(* IEC 61131-3 sources: pandora/pandora/aws-platform-main/aws-platform-main/src/Io, 9 files *)

(* ---- Io.st ---- *)
USING Esab.Io;

NAMESPACE Esab.Io

    CLASS ABSTRACT Input
        VAR PUBLIC
            Id : UINT;
            /// The endianness of the read value.
            /// If this is "little" it will be converted to big for use in the PLC-program
            Endianness : Endianness := Endianness#Big;
        END_VAR

        VAR PROTECTED
            _inputChangedHandler : InputChangedListener;
        END_VAR

        METHOD PUBLIC SetChangedHandler
            VAR_INPUT
                handler : InputChangedListener;
            END_VAR

            _inputChangedHandler := handler;
        END_METHOD

        METHOD PUBLIC ABSTRACT HasChanged : BOOL
        END_METHOD
    END_CLASS

    CLASS Output
        VAR PUBLIC
            /// The endianness that the target value is expected to have by the consumer of the output.
            Endianness : Endianness := Endianness#Big;
        END_VAR
    END_CLASS

    INTERFACE InputChangedListener
        METHOD InputChanged
            VAR_INPUT
                input : REF_TO Input;
            END_VAR
        END_METHOD
    END_INTERFACE

    TYPE
        /// Used in Inputs and Outputs to convert endianness properly.
        /// The PLC uses big endian, while data coming from some outside source may be little.
        Endianness : INT(Big := 0, Little := 1);
    END_TYPE

END_NAMESPACE

(* ---- Digital.st ---- *)
NAMESPACE Esab.Io

    INTERFACE IDigitalInput
        /// Reads a new value
        METHOD Read
            VAR_INPUT
                value : BOOL;
            END_VAR
        END_METHOD

        /// Returns the last value read
        METHOD GetValue : BOOL
        END_METHOD

        /// Returns TRUE if the input experienced a rising edge
        METHOD RisingEdge : BOOL
        END_METHOD

        /// Returns TRUE if the input experienced a falling edge
        METHOD FallingEdge : BOOL
        END_METHOD
    END_INTERFACE

    INTERFACE IDigitalOutput
        /// Writes the value to the output
        METHOD Write
            VAR_OUTPUT
                value : BOOL;
            END_VAR
        END_METHOD

        /// Sets the current value to the given value
        METHOD SetValue
            VAR_INPUT
                value: BOOL;
            END_VAR
        END_METHOD

        /// Sets the current value to TRUE
        METHOD Set
        END_METHOD

        /// Reset the current value to FALSE
        METHOD Reset
        END_METHOD

        /// Toggles the current value
        METHOD Toggle
        END_METHOD
    END_INTERFACE

    CLASS DigitalInput EXTENDS Input IMPLEMENTS IDigitalInput
        VAR PRIVATE
            _currentValue : BOOL;
            _lastValue : BOOL;
        END_VAR

        METHOD PUBLIC Read
            VAR_INPUT
                value : BOOL;
            END_VAR

            _lastValue := _currentValue;
            _currentValue := value;

            IF _inputChangedHandler <> NULL AND THIS.RisingEdge() THEN
                _inputChangedHandler.InputChanged(REF(THIS));
            END_IF;

            IF _inputChangedHandler <> NULL AND THIS.FallingEdge() THEN
                _inputChangedHandler.InputChanged(REF(THIS));
            END_IF;
        END_METHOD

        METHOD PUBLIC GetValue : BOOL
            GetValue := _currentValue;
        END_METHOD

        METHOD PUBLIC RisingEdge : BOOL
            RisingEdge := NOT _lastValue AND _currentValue;
        END_METHOD

        METHOD PUBLIC FallingEdge : BOOL
            FallingEdge := _lastValue AND NOT _currentValue;
        END_METHOD

        METHOD PUBLIC OVERRIDE HasChanged : BOOL
            HasChanged := _lastValue <> _currentValue;
        END_METHOD
    END_CLASS

    CLASS DigitalOutput EXTENDS Output IMPLEMENTS IDigitalOutput
        VAR PRIVATE
            _value : BOOL;
        END_VAR

        METHOD PUBLIC Write
            VAR_OUTPUT
                value : BOOL;
            END_VAR

            value := _value;
        END_METHOD

        METHOD PUBLIC SetValue
            VAR_INPUT
                value: BOOL;
            END_VAR

            _value := value;
        END_METHOD

        METHOD PUBLIC Set
            _value := TRUE;
        END_METHOD

        METHOD PUBLIC Reset
            _value := FALSE;
        END_METHOD

        METHOD PUBLIC Toggle
            _value := NOT _value;
        END_METHOD
    END_CLASS

    CLASS DigitalInOut EXTENDS DigitalInput IMPLEMENTS IDigitalOutput
        VAR PRIVATE
            _value : BOOL;
        END_VAR

        METHOD PUBLIC Write
            VAR_OUTPUT
                value : BOOL;
            END_VAR

            value := _value;
        END_METHOD

        METHOD PUBLIC SetValue
            VAR_INPUT
                value: BOOL;
            END_VAR

            _value := value;
        END_METHOD

        METHOD PUBLIC Set
            _value := TRUE;
        END_METHOD

        METHOD PUBLIC Reset
            _value := FALSE;
        END_METHOD

        METHOD PUBLIC Toggle
            _value := NOT _value;
        END_METHOD
    END_CLASS

END_NAMESPACE

(* ---- DInt.st ---- *)
USING Esab.Utils;

NAMESPACE Esab.Io

    INTERFACE IDIntInput
        /// Reads a new value
        METHOD Read
            VAR_INPUT
                value : DINT;
            END_VAR
        END_METHOD

        /// Returns the last value read
        METHOD GetValue : DINT
        END_METHOD
    END_INTERFACE

    INTERFACE IDIntOutput
        /// Writes the value to the output
        METHOD Write
            VAR_OUTPUT
                value : DINT;
            END_VAR
        END_METHOD

        /// Sets the current value to the given value
        METHOD SetValue
            VAR_INPUT
                value: DINT;
            END_VAR
        END_METHOD
    END_INTERFACE

    CLASS DIntInput EXTENDS Input IMPLEMENTS IDIntInput
        VAR PRIVATE
            _lastValue : DINT;
            _value : DINT;
        END_VAR

        METHOD PUBLIC Read
            VAR_INPUT
                value : DINT;
            END_VAR

            VAR_TEMP
                convertedValue : DINT;
            END_VAR

            convertedValue := value;

            IF THIS.Endianness = Endianness#Little THEN
                convertedValue := TO_DINT(Flip(value));
            END_IF;

            _lastValue := _value;
            _value := convertedValue;

            IF THIS.HasChanged() AND _inputChangedHandler <> NULL THEN
                _inputChangedHandler.InputChanged(REF(THIS));
            END_IF;
        END_METHOD

        METHOD PUBLIC GetValue : DINT
            GetValue := _value;
        END_METHOD

        METHOD PUBLIC OVERRIDE HasChanged : BOOL
            HasChanged := _lastValue <> _value;
        END_METHOD
    END_CLASS

    CLASS DIntOutput EXTENDS Output IMPLEMENTS IDIntOutput
        VAR PRIVATE
            _value : DINT;
        END_VAR

        METHOD PUBLIC Write
            VAR_OUTPUT
                value : DINT;
            END_VAR

            VAR_TEMP
                convertedValue : DINT;
            END_VAR

            convertedValue := _value;

            IF THIS.Endianness = Endianness#Little THEN
                convertedValue := TO_DINT(Flip(_value));
            END_IF;

            value := convertedValue;
        END_METHOD

        METHOD PUBLIC SetValue
            VAR_INPUT
                value: DINT;
            END_VAR

            _value := value;
        END_METHOD
    END_CLASS

END_NAMESPACE

(* ---- HighSpeedCounter.st ---- *)
USING Esab.Io;
USING Esab.Utils.Alarming;

NAMESPACE Esab.Io

    /// Interface for a HSC wrapper.
    INTERFACE IHighSpeedCounter
        /// Cyclic execute.
        METHOD Execute
        END_METHOD

        /// Enables the counter
        METHOD Enable
        END_METHOD

        /// Disables the counter
        METHOD Disable
        END_METHOD

        /// Returns the counter value in increments
        METHOD GetCountValue : DINT
        END_METHOD

        /// Returns the measured value, for our application this is the speed
        /// in increments/second
        METHOD GetMeasuredValue : DINT
        END_METHOD

        /// Returns the maximum possible value for this counter
        METHOD GetUpperCountingLimit : DINT
        END_METHOD

        /// Returns the minimum possible value for this counter
        METHOD GetLowerCountingLimit : DINT
        END_METHOD

        /// Reset counter value to value
        METHOD SetCountValue
            VAR_INPUT
                value : DINT;
            END_VAR
        END_METHOD

        /// Returns TRUE if the counter has an error.
        METHOD HasError : BOOL
        END_METHOD
    END_INTERFACE

    CLASS HighSpeedCounter EXTENDS Object IMPLEMENTS IHighSpeedCounter, InputChangedListener
        VAR PRIVATE
            _io : REF_TO HighSpeedCounterIo;
            _hardwareConfiguration : REF_TO HighSpeedCounterHardwareConfiguration;
            _loadCommandErrorAlarm : IAlarm;
            _encoderErrorAlarm : IAlarm;
            _powerSupplyAlarm : IAlarm;

            _currentSlot0Command : HighSpeedCounterLoadCommand;
            _currentSlot1Command : HighSpeedCounterLoadCommand;
        END_VAR

        METHOD PUBLIC Setup
            VAR_INPUT
                io : REF_TO HighSpeedCounterIo;
                hardwareConfiguration : REF_TO HighSpeedCounterHardwareConfiguration;
                loadCommandErrorAlarm : IAlarm;
                encoderErrorAlarm : IAlarm;
                powerSupplyAlarm : IAlarm;
                setupAlarm : IAlarm;
            END_VAR

            _io := io;
            _hardwareConfiguration := hardwareConfiguration;
            _loadCommandErrorAlarm := loadCommandErrorAlarm;
            _encoderErrorAlarm := encoderErrorAlarm;
            _powerSupplyAlarm := powerSupplyAlarm;
            _setupAlarm := setupAlarm;

            _isSetup := _io <> NULL AND _hardwareConfiguration <> NULL AND _encoderErrorAlarm <> NULL AND _powerSupplyAlarm <> NULL;

            IF _isSetup THEN
                _io^.Inputs.LoadError.SetChangedHandler(THIS);
                _io^.Inputs.Slot0Loaded.SetChangedHandler(THIS);
                _io^.Inputs.Slot1Loaded.SetChangedHandler(THIS);

                THIS.LoadSlot0(_hardwareConfiguration^.LowerCountingLimit, HighSpeedCounterLoadCommand#LoadLowCountingLimit);
                THIS.LoadSlot1(_hardwareConfiguration^.UpperCountingLimit, HighSpeedCounterLoadCommand#LoadHighCountingLimit);
            END_IF;
        END_METHOD

        METHOD PUBLIC OVERRIDE Execute
            SUPER.Execute();

            IF _setupAlarm.IsActive() THEN
                RETURN;
            END_IF;

            _loadCommandErrorAlarm.Execute(_io^.Inputs.LoadError.GetValue());
            _encoderErrorAlarm.Execute(_io^.Inputs.EncoderError.GetValue());
            _powerSupplyAlarm.Execute(_io^.Inputs.PowerSupplyError.GetValue());
        END_METHOD

        METHOD PUBLIC OVERRIDE UpdateState
            IF _setupAlarm.IsActive() THEN
                _currentState := HighSpeedCounterState#Error;
            ELSIF _encoderErrorAlarm.IsActive() OR _powerSupplyAlarm.IsActive() THEN
                _currentState := HighSpeedCounterState#Error;
            ELSE
                _currentState := HighSpeedCounterState#Healthy;
            END_IF;
        END_METHOD

        METHOD PUBLIC SetHardwareConfiguration
            VAR_INPUT
                hwConfiguration : REF_TO HighSpeedCounterHardwareConfiguration;
            END_VAR

            _hardwareConfiguration := hwConfiguration;
        END_METHOD

        METHOD PUBLIC Enable
            _io^.Outputs.SoftwareGate.Set();
        END_METHOD

        METHOD PUBLIC Disable
            _io^.Outputs.SoftwareGate.Reset();
        END_METHOD

        METHOD PUBLIC GetCountValue : DINT
            GetCountValue := _io^.Inputs.CountValue.GetValue();
        END_METHOD

        METHOD PUBLIC GetMeasuredValue : DINT
            GetMeasuredValue := _io^.Inputs.MeasuredValue.GetValue();
        END_METHOD

        METHOD PUBLIC GetUpperCountingLimit : DINT
            GetUpperCountingLimit := _hardwareConfiguration^.UpperCountingLimit;
        END_METHOD

        METHOD PUBLIC GetLowerCountingLimit : DINT
            GetLowerCountingLimit := _hardwareConfiguration^.LowerCountingLimit;
        END_METHOD

        METHOD PUBLIC SetCountValue
            VAR_INPUT
                value : DINT;
            END_VAR

            _io^.Outputs.Slot0.SetValue(value);
            _io^.Outputs.LoadSlotX.SetValue(HighSpeedCounterLoadCommand#LoadCounter);
        END_METHOD

        METHOD PUBLIC HasError : BOOL
            HasError := THIS.GetState() = HighSpeedCounterState#Error;
        END_METHOD

        METHOD PUBLIC InputChanged
            VAR_INPUT
                input : REF_TO Esab.Io.Input;
            END_VAR

            IF (input = REF(_io^.Inputs.LoadError) AND _io^.Inputs.LoadError.RisingEdge()) OR
               (input = REF(_io^.Inputs.Slot0Loaded) AND _io^.Inputs.Slot0Loaded.RisingEdge()) THEN

                THIS.LoadSlot0(DINT#0, HighSpeedCounterLoadCommand#Idle);
            ELSIF (input = REF(_io^.Inputs.LoadError) AND _io^.Inputs.LoadError.RisingEdge()) OR
                  (input = REF(_io^.Inputs.Slot0Loaded) AND _io^.Inputs.Slot0Loaded.RisingEdge()) THEN

                THIS.LoadSlot1(DINT#0, HighSpeedCounterLoadCommand#Idle);
            END_IF;
        END_METHOD

        METHOD PRIVATE LoadSlot0
            VAR_INPUT
                value : DINT;
                command : HighSpeedCounterLoadCommand;
            END_VAR

            _io^.Outputs.Slot0.SetValue(value);
            _currentSlot0Command := command;
            _io^.Outputs.LoadSlotX.SetValue(_currentSlot0Command AND SHL(_currentSlot1Command, UINT#4));
        END_METHOD

        METHOD PRIVATE LoadSlot1
            VAR_INPUT
                value : DINT;
                command : HighSpeedCounterLoadCommand;
            END_VAR

            _io^.Outputs.Slot1.SetValue(value);
            _currentSlot1Command := command;
            _io^.Outputs.LoadSlotX.SetValue(_currentSlot0Command AND SHL(_currentSlot1Command, UINT#4));
        END_METHOD
    END_CLASS

    TYPE
        HighSpeedCounterHardwareConfiguration : STRUCT
            UpperCountingLimit : DINT := DINT#2147483647;
            LowerCountingLimit : DINT := DINT#-2147483648;
        END_STRUCT;

        HighSpeedCounterState : INT(
            Healthy := 0,
            Error := 1
        );

        HighSpeedCounterLoadCommand : BYTE(
            Idle := BYTE#0,
            LoadCounter := BYTE#1,
            LoadStartValue := BYTE#3,
            LoadComparison0 := BYTE#4,
            LoadComparison1 := BYTE#5,
            LoadLowCountingLimit := BYTE#6,
            LoadHighCountingLimit := BYTE#7
        );

        HighSpeedCounterIo : STRUCT
            Inputs : HighSpeedCounterInputs;
            Outputs : HighSpeedCounterOutputs;
        END_STRUCT;

        HighSpeedCounterOutputs : STRUCT
            Slot0 : DIntOutput;
            Slot1 : DIntOutput;
            LoadSlotX : UIntOutput;
            EnableCapture : DigitalOutput;
            EnableSynchronizationDown : DigitalOutput;
            EnableSynchronizationUp : DigitalOutput;
            SetDq1 : DigitalOutput;
            SetDq0 : DigitalOutput;
            TmCtrlDq1 : DigitalOutput;
            TmCtrlDq0 : DigitalOutput;
            SoftwareGate : DigitalOutput;
            CountDirection : DigitalOutput;
            ResetEvents : DigitalOutput;
            ResetErrors : DigitalOutput;
        END_STRUCT;

        HighSpeedCounterInputs : STRUCT
            CountValue : DIntInput;
            CapturedValue : DIntInput;
            MeasuredValue : DIntInput;
            LoadError : DigitalInput;
            EncoderError : DigitalInput;
            PowerSupplyError : DigitalInput;
            SoftwareGate : DigitalInput;
            Ready : DigitalInput;
            Slot1Loaded : DigitalInput;
            Slot0Loaded : DigitalInput;
            ResetEventsAcknowledge : DigitalInput;
            Di2 : DigitalInput;
            Di1 : DigitalInput;
            Di0 : DigitalInput;
            Dq1 : DigitalInput;
            Dq0 : DigitalInput;
            InternalGate : DigitalInput;
            Counting : DigitalInput;
            Direction : DigitalInput;
            MeasurementPulseDetected : DigitalInput;
            CaptureEvent : DigitalInput;
            SynchronizationEvent : DigitalInput;
            ComparisonEvent1 : DigitalInput;
            ComparisonEvent0 : DigitalInput;
            OverflowEvent : DigitalInput;
            UnderflowEvent : DigitalInput;
            ZeroPassEvent : DigitalInput;
        END_STRUCT;

        RawHighSpeedCounterOutputs : STRUCT
            Slot0 AT %B0 : DINT;
            Slot1 AT %B4 : DINT;
            LoadSlotX AT %B8 : BYTE;
            EnableCapture AT %X9.7 : BOOL;
            EnableSynchronizationDown AT %X9.6 : BOOL;
            EnableSynchronizationUp AT %X9.5 : BOOL;
            SetDq1 AT %X9.4 : BOOL;
            SetDq0 AT %X9.3 : BOOL;
            TmCtrlDq1 AT %X9.2 : BOOL;
            TmCtrlDq0 AT %X9.1 : BOOL;
            SoftwareGate AT %X9.0 : BOOL;
            CountDirection AT %X10.7 : BOOL;
            // Bits 2 to 6 are reserved
            ResetEvents AT %X10.1 : BOOL;
            ResetErrors AT %X10.0 : BOOL;
        END_STRUCT;

        RawHighSpeedCounterInputs : STRUCT
            CountValue AT %B0 : DINT;
            CapturedValue AT %B4 : DINT;
            MeasuredValue AT %B8 : DINT;
            // Bits 2 to 7 are reserved
            LoadError AT %X12.2 : BOOL;
            EncoderError AT %X12.1 : BOOL;
            PowerSupplyError AT %X12.0 : BOOL;
            // Bits 6 to 7 are reserved
            SoftwareGate AT %X13.5 : BOOL;
            Ready AT %X13.4 : BOOL;
            Slot1Loaded AT %X13.3 : BOOL;
            Slot0Loaded AT %X13.2 : BOOL;
            ResetEventsAcknowledge AT %X13.1 : BOOL;
            // Bit 0 is reserved
            Di2 AT %X14.7 : BOOL;
            Di1 AT %X14.6 : BOOL;
            Di0 AT %X14.5 : BOOL;
            Dq1 AT %X14.4 : BOOL;
            Dq0 AT %X14.3 : BOOL;
            InternalGate AT %X14.2 : BOOL;
            Counting AT %X14.1 : BOOL;
            Direction AT %X14.0 : BOOL;
            MeasurementPulseDetected AT %X15.7 : BOOL;
            CaptureEvent AT %X15.6 : BOOL;
            SynchronizationEvent AT %X15.5 : BOOL;
            ComparisonEvent1 AT %X15.4 : BOOL;
            ComparisonEvent0 AT %X15.3 : BOOL;
            OverflowEvent AT %X15.2 : BOOL;
            UnderflowEvent AT %X15.1 : BOOL;
            ZeroPassEvent AT %X15.0 : BOOL;
        END_STRUCT;
    END_TYPE

END_NAMESPACE

(* ---- Int.st ---- *)
USING Esab.Utils;

NAMESPACE Esab.Io

    INTERFACE IIntInput
        /// Reads a new value
        METHOD Read
            VAR_INPUT
                value : INT;
            END_VAR
        END_METHOD

        /// Returns the last value read
        METHOD GetValue : INT
        END_METHOD
    END_INTERFACE

    INTERFACE IIntOutput
        /// Writes the value to the output
        METHOD Write
            VAR_OUTPUT
                value : INT;
            END_VAR
        END_METHOD

        /// Sets the current value to the given value
        METHOD SetValue
            VAR_INPUT
                value: INT;
            END_VAR
        END_METHOD
    END_INTERFACE

    CLASS IntInput EXTENDS Input IMPLEMENTS IIntInput
        VAR PRIVATE
            _lastValue : INT;
            _value : INT;
        END_VAR

        METHOD PUBLIC Read
            VAR_INPUT
                value : INT;
            END_VAR

            VAR_TEMP
                convertedValue : INT;
            END_VAR

            convertedValue := value;

            IF THIS.Endianness = Endianness#Little THEN
                convertedValue := TO_INT(Flip(value));
            END_IF;

            _lastValue := _value;
            _value := convertedValue;

            IF THIS.HasChanged() AND _inputChangedHandler <> NULL THEN
                _inputChangedHandler.InputChanged(REF(THIS));
            END_IF;
        END_METHOD

        METHOD PUBLIC GetValue : INT
            GetValue := _value;
        END_METHOD

        METHOD PUBLIC OVERRIDE HasChanged : BOOL
            HasChanged := _lastValue <> _value;
        END_METHOD
    END_CLASS

    CLASS IntOutput EXTENDS Output IMPLEMENTS IIntOutput

        VAR PRIVATE
            _value : INT;
        END_VAR

        METHOD PUBLIC Write
            VAR_OUTPUT
                value : INT;
            END_VAR

            VAR_TEMP
                convertedValue : INT;
            END_VAR

            convertedValue := _value;

            IF THIS.Endianness = Endianness#Little THEN
                convertedValue := TO_INT(Flip(_value));
            END_IF;

            value := convertedValue;
        END_METHOD

        METHOD PUBLIC SetValue
            VAR_INPUT
                value: INT;
            END_VAR

            _value := value;
        END_METHOD
    END_CLASS

END_NAMESPACE

(* ---- Real.st ---- *)
USING Esab.Utils;

USING System.FastMath;

NAMESPACE Esab.Io

    INTERFACE IRealInput
        /// Reads a new value
        /// The value will be read, and scaling applied.
        METHOD Read
            VAR_INPUT
                value : REAL;
            END_VAR
        END_METHOD

        /// Reads a new value (DWORD)
        /// Here it is assumed that the DWORD bytes are representing a REAL
        METHOD Read
            VAR_INPUT
                value : DWORD;
            END_VAR
        END_METHOD

        /// Reads a new value (UINT)
        /// The value will be read, converted to real, and scaling applied.
        METHOD Read
            VAR_INPUT
                value : UINT;
            END_VAR
        END_METHOD

        /// Reads a new value (INT)
        /// The value will be read, converted to real, and scaling applied.
        METHOD Read
            VAR_INPUT
                value : INT;
            END_VAR
        END_METHOD

        /// Returns the last value read
        METHOD GetValue : REAL
        END_METHOD
    END_INTERFACE

    INTERFACE IRealOutput
        /// Writes the value to the output
        METHOD Write
            VAR_OUTPUT
                value : REAL;
            END_VAR
        END_METHOD

        /// Writes the value to the output (DWORD)
        METHOD Write
            VAR_OUTPUT
                value : DWORD;
            END_VAR
        END_METHOD

        /// Writes the value to the output (INT)
        METHOD Write
            VAR_OUTPUT
                value : INT;
            END_VAR
        END_METHOD

        /// Sets the current value to the given value
        METHOD SetValue
            VAR_INPUT
                value: REAL;
            END_VAR
        END_METHOD
    END_INTERFACE

    CLASS RealInput EXTENDS Input IMPLEMENTS IRealInput
        VAR PUBLIC
            /// Delta used when deciding if this input has changed
            ChangeDelta : REAL := REAL#0.01;
            /// Scaling will be applied when reading the input
            /// E.g. if the input read is a DINT with the unit 0.1 radishes, a scale of 0.1 will result in GetValue() returning a
            /// REAL with the unit 1.0 radishes, so input = DINT#2 -> GetValue() = 0.2 radishes.
            Scale : REAL := REAL#1.0;
        END_VAR

        VAR PRIVATE
            _lastValue : REAL;
            _value : REAL;
        END_VAR

        METHOD PUBLIC Read
            VAR_INPUT
                value : REAL;
            END_VAR

            VAR_TEMP
                convertedValue : REAL;
            END_VAR

            convertedValue := value;

            IF endianness = Endianness#Little THEN
                convertedValue := TO_REAL(Flip(value));
            END_IF;

            _lastValue := _value;
            _value := convertedValue * THIS.Scale;

            IF THIS.HasChanged() AND _inputChangedHandler <> NULL THEN
                _inputChangedHandler.InputChanged(REF(THIS));
            END_IF;
        END_METHOD

        METHOD PUBLIC Read
            VAR_INPUT
                value : DWORD;
            END_VAR

            VAR_TEMP
                convertedValue : REAL;
            END_VAR

            convertedValue := TO_REAL(value);

            IF THIS.Endianness = Endianness#Little THEN
                convertedValue := TO_REAL(Flip(value));
            END_IF;

            _lastValue := _value;
            _value := convertedValue * THIS.Scale;

            IF THIS.HasChanged() AND _inputChangedHandler <> NULL THEN
                _inputChangedHandler.InputChanged(REF(THIS));
            END_IF;
        END_METHOD

        METHOD PUBLIC Read
            VAR_INPUT
                value : UINT;
            END_VAR

            VAR_TEMP
                convertedValue : REAL;
            END_VAR

            convertedValue := TO_REAL(value);

            IF THIS.Endianness = Endianness#Little THEN
                convertedValue := TO_REAL(Flip(TO_REAL(value)));
            END_IF;

            _lastValue := _value;
            _value := convertedValue * THIS.Scale;

            IF THIS.HasChanged() AND _inputChangedHandler <> NULL THEN
                _inputChangedHandler.InputChanged(REF(THIS));
            END_IF;
        END_METHOD

        METHOD PUBLIC Read
            VAR_INPUT
                value : INT;
            END_VAR

            VAR_TEMP
                convertedValue : REAL;
            END_VAR

            convertedValue := value;

            IF THIS.Endianness = Endianness#Little THEN
                convertedValue := TO_REAL(Flip(TO_REAL(value)));
            END_IF;

            _lastValue := _value;
            _value := convertedValue * THIS.Scale;

            IF THIS.HasChanged() AND _inputChangedHandler <> NULL THEN
                _inputChangedHandler.InputChanged(REF(THIS));
            END_IF;
        END_METHOD

        METHOD PUBLIC GetValue : REAL
            GetValue := _value;
        END_METHOD

        METHOD PUBLIC OVERRIDE HasChanged : BOOL
            HasChanged := ABS(_lastValue - _value) > ChangeDelta;
        END_METHOD
    END_CLASS

    /// Implements a normalized real input.
    /// If bipolar = TRUE then the value in the range [Minimum, Maximum] will be normalized to [-1.0, 1.0]
    /// If bipolar = FALSE then the value in the range [Minimum, Maximum] will be normalized to [0.0, 1.0] (this is the default)
    CLASS RealNormalizedInput EXTENDS Input IMPLEMENTS IRealInput
        VAR PUBLIC
            /// Delta used when deciding if this input has changed
            ChangeDelta : REAL := REAL#0.01;
            /// If this is a bipolar input or not
            Bipolar : BOOL := FALSE;
            /// Minimum possible input value
            Minimum : REAL := REAL#0.0;
            /// Maximum possible input value
            Maximum : REAL := REAL#27648.0;
        END_VAR

        VAR PRIVATE
            _lastValue : REAL;
            _value : REAL;
        END_VAR

        METHOD PUBLIC Read
            VAR_INPUT
                value : REAL;
            END_VAR

            VAR_TEMP
                convertedValue : REAL;
            END_VAR

            convertedValue := value;

            IF endianness = Endianness#Little THEN
                convertedValue := TO_REAL(Flip(value));
            END_IF;

            convertedValue := THIS.Normalize(convertedValue);

            _lastValue := _value;
            _value := convertedValue;

            IF THIS.HasChanged() AND _inputChangedHandler <> NULL THEN
                _inputChangedHandler.InputChanged(REF(THIS));
            END_IF;
        END_METHOD

        METHOD PUBLIC Read
            VAR_INPUT
                value : DWORD;
            END_VAR

            VAR_TEMP
                convertedValue : REAL;
            END_VAR

            convertedValue := TO_REAL(value);

            IF endianness = Endianness#Little THEN
                convertedValue := TO_REAL(Flip(value));
            END_IF;

            convertedValue := THIS.Normalize(convertedValue);

            _lastValue := _value;
            _value := convertedValue;

            IF THIS.HasChanged() AND _inputChangedHandler <> NULL THEN
                _inputChangedHandler.InputChanged(REF(THIS));
            END_IF;
        END_METHOD

        METHOD PUBLIC Read
            VAR_INPUT
                value : UINT;
            END_VAR

            VAR_TEMP
                convertedValue : REAL;
            END_VAR

            convertedValue := TO_REAL(value);

            IF endianness = Endianness#Little THEN
                convertedValue := TO_REAL(Flip(TO_REAL(value)));
            END_IF;

            convertedValue := THIS.Normalize(convertedValue);

            _lastValue := _value;
            _value := convertedValue;

            IF THIS.HasChanged() AND _inputChangedHandler <> NULL THEN
                _inputChangedHandler.InputChanged(REF(THIS));
            END_IF;
        END_METHOD

        METHOD PUBLIC Read
            VAR_INPUT
                value : INT;
            END_VAR

            VAR_TEMP
                convertedValue : REAL;
            END_VAR

            convertedValue := TO_REAL(value);

            IF endianness = Endianness#Little THEN
                convertedValue := TO_REAL(Flip(TO_REAL(value)));
            END_IF;

            convertedValue := THIS.Normalize(convertedValue);

            _lastValue := _value;
            _value := convertedValue;

            IF THIS.HasChanged() AND _inputChangedHandler <> NULL THEN
                _inputChangedHandler.InputChanged(REF(THIS));
            END_IF;
        END_METHOD

        METHOD PUBLIC GetValue : REAL
            GetValue := _value;
        END_METHOD

        METHOD PUBLIC OVERRIDE HasChanged : BOOL
            HasChanged := ABS(_lastValue - _value) > ChangeDelta;
        END_METHOD

        METHOD PRIVATE Normalize : REAL
            VAR_INPUT
                value : REAL;
            END_VAR

            VAR_TEMP
                _normalized : REAL;
            END_VAR

            IF THIS.Bipolar THEN
                _normalized := (value - THIS.Minimum) / (THIS.Maximum - THIS.Minimum) * REAL#2.0 - REAL#1.0;
            ELSE
                _normalized := (value - THIS.Minimum) / (THIS.Maximum - THIS.Minimum);
            END_IF;

            Normalize := _normalized;
        END_METHOD
    END_CLASS

    CLASS RealOutput EXTENDS Output IMPLEMENTS IRealOutput
        VAR PUBLIC
            /// Scaling will be applied when writing the output
            /// E.g. if the output written is a DINT with the unit 0.1 radishes, a scale of 0.1 will result in Write() outputting
            /// a number with the unit 0.1 radishes, so SetValue(REAL#0.2) -> output = DINT#2 radishes.
            Scale : REAL := REAL#1.0;
        END_VAR

        VAR PRIVATE
            _value : REAL;
        END_VAR

        METHOD PUBLIC Write
            VAR_OUTPUT
                value : REAL;
            END_VAR

            VAR_TEMP
                convertedValue : REAL;
            END_VAR

            convertedValue := _value / THIS.Scale;

            IF THIS.Endianness = Endianness#Little THEN
                convertedValue := TO_REAL(Flip(convertedValue));
            END_IF;

            value := convertedValue;
        END_METHOD

        METHOD PUBLIC Write
            VAR_OUTPUT
                value : DWORD;
            END_VAR

            VAR_TEMP
                convertedValue : DWORD;
            END_VAR

            convertedValue := TO_DWORD(_value / THIS.Scale);

            IF THIS.Endianness = Endianness#Little THEN
                convertedValue := Flip(convertedValue);
            END_IF;

            value := convertedValue;
        END_METHOD

        METHOD PUBLIC Write
            VAR_OUTPUT
                value : UINT;
            END_VAR

            VAR_TEMP
                convertedValue : UINT;
            END_VAR

            convertedValue := TO_UINT(_value / THIS.Scale);

            IF THIS.Endianness = Endianness#Little THEN
                convertedValue := TO_UINT(Flip(convertedValue));
            END_IF;

            value := convertedValue;
        END_METHOD

        METHOD PUBLIC Write
            VAR_OUTPUT
                value : INT;
            END_VAR

            VAR_TEMP
                convertedValue : INT;
            END_VAR

            convertedValue := TO_INT(_value / THIS.Scale);

            IF THIS.Endianness = Endianness#Little THEN
                convertedValue := TO_INT(Flip(convertedValue));
            END_IF;

            value := convertedValue;
        END_METHOD

        METHOD PUBLIC SetValue
            VAR_INPUT
                value: REAL;
            END_VAR

            _value := value;
        END_METHOD
    END_CLASS

    CLASS RealNormalizedOutput EXTENDS Output IMPLEMENTS IRealOutput
        VAR PUBLIC
            /// If this is a bipolar output or not
            Bipolar : BOOL := FALSE;
            /// Minimum possible output value
            Minimum : REAL := REAL#0.0;
            /// Maximum possible output value
            Maximum : REAL := REAL#27648.0;
        END_VAR

        VAR PRIVATE
            _value : REAL;
        END_VAR

        METHOD PUBLIC Write
            VAR_OUTPUT
                value : REAL;
            END_VAR

            VAR_TEMP
                convertedValue : REAL;
            END_VAR

            convertedValue := THIS.Normalize(_value);

            IF THIS.Endianness = Endianness#Little THEN
                convertedValue := TO_REAL(Flip(convertedValue));
            END_IF;

            value := convertedValue;
        END_METHOD

        METHOD PUBLIC Write
            VAR_OUTPUT
                value : DWORD;
            END_VAR

            VAR_TEMP
                convertedValue : DWORD;
            END_VAR

            convertedValue := TO_DWORD(THIS.Normalize(_value));

            IF THIS.Endianness = Endianness#Little THEN
                convertedValue := Flip(convertedValue);
            END_IF;

            value := convertedValue;
        END_METHOD

        METHOD PUBLIC Write
            VAR_OUTPUT
                value : UINT;
            END_VAR

            VAR_TEMP
                convertedValue : UINT;
            END_VAR

            convertedValue := TO_UINT(THIS.Normalize(_value));

            IF THIS.Endianness = Endianness#Little THEN
                convertedValue := TO_UINT(Flip(convertedValue));
            END_IF;

            value := convertedValue;
        END_METHOD

        METHOD PUBLIC Write
            VAR_OUTPUT
                value : INT;
            END_VAR

            VAR_TEMP
                convertedValue : INT;
            END_VAR

            convertedValue := TO_INT(THIS.Normalize(_value));

            IF THIS.Endianness = Endianness#Little THEN
                convertedValue := TO_INT(Flip(convertedValue));
            END_IF;

            value := convertedValue;
        END_METHOD

        METHOD PUBLIC SetValue
            VAR_INPUT
                value: REAL;
            END_VAR

            _value := value;

            IF value > 1.0 THEN
                _value := REAL#1.0;
            ELSIF Bipolar && value < -1.0 THEN
                _value := REAL#-1.0;
            ELSIF NOT Bipolar && value < 0.0 THEN
                _value := REAL#0.0;
            END_IF;
        END_METHOD

        METHOD PRIVATE Normalize : REAL
            VAR_INPUT
                value : REAL;
            END_VAR

            VAR_TEMP
                _normalized : REAL;
            END_VAR

            IF THIS.Bipolar THEN
                _normalized := (value + REAL#1.0) / REAL#2.0 * (THIS.Maximum - THIS.Minimum) + THIS.Minimum;
            ELSE
                _normalized := value * (THIS.Maximum - THIS.Minimum) + THIS.Minimum;
            END_IF;

            Normalize := _normalized;
        END_METHOD
    END_CLASS

END_NAMESPACE

(* ---- UDInt.st ---- *)
USING Esab.Utils;

NAMESPACE Esab.Io

    INTERFACE IUDIntInput
        /// Reads a new value
        METHOD Read
            VAR_INPUT
                value : UDINT;
            END_VAR
        END_METHOD

        /// Returns the last value read
        METHOD GetValue : UDINT
        END_METHOD
    END_INTERFACE

    INTERFACE IUDIntOutput
        /// Writes the value to the output
        METHOD Write
            VAR_OUTPUT
                value : UDINT;
            END_VAR
        END_METHOD

        /// Sets the current value to the given value
        METHOD SetValue
            VAR_INPUT
                value: UDINT;
            END_VAR
        END_METHOD
    END_INTERFACE

    CLASS UDIntInput EXTENDS Input IMPLEMENTS IUDIntInput
        VAR PRIVATE
            _lastValue : UDINT;
            _value : UDINT;
        END_VAR

        METHOD PUBLIC Read
            VAR_INPUT
                value : UDINT;
            END_VAR

            VAR_TEMP
                convertedValue : UDINT;
            END_VAR

            convertedValue := value;

            IF THIS.Endianness = Endianness#Little THEN
                convertedValue := TO_UDINT(Flip(value));
            END_IF;

            _lastValue := _value;
            _value := convertedValue;

            IF THIS.HasChanged() AND _inputChangedHandler <> NULL THEN
                _inputChangedHandler.InputChanged(REF(THIS));
            END_IF;
        END_METHOD

        METHOD PUBLIC GetValue : UDINT
            GetValue := _value;
        END_METHOD

        METHOD PUBLIC OVERRIDE HasChanged : BOOL
            HasChanged := _lastValue <> _value;
        END_METHOD
    END_CLASS

    CLASS UDIntOutput EXTENDS Output IMPLEMENTS IUDIntOutput
        VAR PRIVATE
            _value : UDINT;
        END_VAR

        METHOD PUBLIC Write
            VAR_OUTPUT
                value : UDINT;
            END_VAR

            VAR_TEMP
                convertedValue : UDINT;
            END_VAR

            convertedValue := _value;

            IF THIS.Endianness = Endianness#Little THEN
                convertedValue := TO_UDINT(Flip(_value));
            END_IF;

            value := convertedValue;
        END_METHOD

        METHOD PUBLIC SetValue
            VAR_INPUT
                value: UDINT;
            END_VAR

            _value := value;
        END_METHOD
    END_CLASS

END_NAMESPACE

(* ---- UInt.st ---- *)
USING Esab.Utils;

NAMESPACE Esab.Io

    INTERFACE IUIntInput
        /// Reads a new value
        METHOD Read
            VAR_INPUT
                value : UINT;
            END_VAR
        END_METHOD

        /// Reads a new value (BYTE)
        METHOD Read
            VAR_INPUT
                value : BYTE;
            END_VAR
        END_METHOD

        /// Returns the last value read
        METHOD GetValue : UINT
        END_METHOD
    END_INTERFACE

    INTERFACE IUIntOutput
        /// Writes the value to the output
        METHOD Write
            VAR_OUTPUT
                value : UINT;
            END_VAR
        END_METHOD

        /// Writes the value to the output (BYTE overload)
        METHOD Write
            VAR_OUTPUT
                value : BYTE;
            END_VAR
        END_METHOD

        /// Sets the current value to the given value
        METHOD SetValue
            VAR_INPUT
                value: UINT;
            END_VAR
        END_METHOD

        /// Sets the current value to the given value (BYTE)
        METHOD SetValue
            VAR_INPUT
                value: BYTE;
            END_VAR
        END_METHOD
    END_INTERFACE

    CLASS UIntInput EXTENDS Input IMPLEMENTS IUIntInput
        VAR PRIVATE
            _lastValue : UINT;
            _value : UINT;
        END_VAR

        METHOD PUBLIC Read
            VAR_INPUT
                value : UINT;
            END_VAR

            VAR_TEMP
                convertedValue : UINT;
            END_VAR

            convertedValue := value;

            IF THIS.Endianness = Endianness#Little THEN
                convertedValue := TO_UINT(Flip(value));
            END_IF;

            _lastValue := _value;
            _value := convertedValue;

            IF THIS.HasChanged() AND _inputChangedHandler <> NULL THEN
                _inputChangedHandler.InputChanged(REF(THIS));
            END_IF;
        END_METHOD

        METHOD PUBLIC Read
            VAR_INPUT
                value : BYTE;
            END_VAR

            VAR_TEMP
                convertedValue : UINT := UINT#0;
            END_VAR

            convertedValue.%B0 := value;

            _lastValue := _value;
            _value := convertedValue;

            IF THIS.HasChanged() AND _inputChangedHandler <> NULL THEN
                _inputChangedHandler.InputChanged(REF(THIS));
            END_IF;
        END_METHOD

        METHOD PUBLIC GetValue : UINT
            GetValue := _value;
        END_METHOD

        METHOD PUBLIC OVERRIDE HasChanged : BOOL
            HasChanged := _lastValue <> _value;
        END_METHOD
    END_CLASS

    CLASS UIntOutput EXTENDS Output IMPLEMENTS IUIntOutput

        VAR PRIVATE
            _value : UINT;
        END_VAR

        METHOD PUBLIC Write
            VAR_OUTPUT
                value : UINT;
            END_VAR

            VAR_TEMP
                convertedValue : UINT;
            END_VAR

            convertedValue := _value;

            IF THIS.Endianness = Endianness#Little THEN
                convertedValue := TO_UINT(Flip(_value));
            END_IF;

            value := convertedValue;
        END_METHOD

        METHOD PUBLIC Write
            VAR_OUTPUT
                value : BYTE;
            END_VAR

            value := _value.%B0;
        END_METHOD

        METHOD PUBLIC SetValue
            VAR_INPUT
                value: UINT;
            END_VAR

            _value := value;
        END_METHOD

        METHOD PUBLIC SetValue
            VAR_INPUT
                value: BYTE;
            END_VAR

            _value := UINT#0;
            _value.%B0 := value;
        END_METHOD
    END_CLASS

END_NAMESPACE

(* ---- Word.st ---- *)
USING Esab.Utils;

NAMESPACE Esab.Io

    INTERFACE IWordInput
        /// Reads a new value
        METHOD Read
            VAR_INPUT
                value : WORD;
            END_VAR
        END_METHOD

        /// Reads a new value (BYTE)
        METHOD Read
            VAR_INPUT
                value : BYTE;
            END_VAR
        END_METHOD

        /// Returns the last value read
        METHOD GetValue : WORD
        END_METHOD
    END_INTERFACE

    INTERFACE IWordOutput
        /// Writes the value to the output
        METHOD Write
            VAR_OUTPUT
                value : WORD;
            END_VAR
        END_METHOD

        /// Writes the value to the output (BYTE overload)
        METHOD Write
            VAR_OUTPUT
                value : BYTE;
            END_VAR
        END_METHOD

        /// Sets the current value to the given value
        METHOD SetValue
            VAR_INPUT
                value: WORD;
            END_VAR
        END_METHOD

        /// Sets the current value to the given value (BYTE)
        METHOD SetValue
            VAR_INPUT
                value: BYTE;
            END_VAR
        END_METHOD
    END_INTERFACE

    CLASS WordInput EXTENDS Input IMPLEMENTS IWordInput
        VAR PRIVATE
            _lastValue : WORD;
            _value : WORD;
        END_VAR

        METHOD PUBLIC Read
            VAR_INPUT
                value : WORD;
            END_VAR

            VAR_TEMP
                convertedValue : WORD;
            END_VAR

            convertedValue := value;

            IF THIS.Endianness = Endianness#Little THEN
                convertedValue := Flip(value);
            END_IF;

            _lastValue := _value;
            _value := convertedValue;

            IF THIS.HasChanged() AND _inputChangedHandler <> NULL THEN
                _inputChangedHandler.InputChanged(REF(THIS));
            END_IF;
        END_METHOD

        METHOD PUBLIC Read
            VAR_INPUT
                value : BYTE;
            END_VAR

            VAR_TEMP
                convertedValue : WORD := WORD#0;
            END_VAR

            convertedValue.%B0 := value;

            _lastValue := _value;
            _value := convertedValue;

            IF THIS.HasChanged() AND _inputChangedHandler <> NULL THEN
                _inputChangedHandler.InputChanged(REF(THIS));
            END_IF;
        END_METHOD

        METHOD PUBLIC GetValue : WORD
            GetValue := _value;
        END_METHOD

        METHOD PUBLIC OVERRIDE HasChanged : BOOL
            HasChanged := _lastValue <> _value;
        END_METHOD
    END_CLASS

    CLASS WordOutput EXTENDS Output IMPLEMENTS IWordOutput

        VAR PRIVATE
            _value : WORD;
        END_VAR

        METHOD PUBLIC Write
            VAR_OUTPUT
                value : WORD;
            END_VAR

            VAR_TEMP
                convertedValue : WORD;
            END_VAR

            convertedValue := _value;

            IF THIS.Endianness = Endianness#Little THEN
                convertedValue := Flip(_value);
            END_IF;

            value := convertedValue;
        END_METHOD

        METHOD PUBLIC Write
            VAR_OUTPUT
                value : BYTE;
            END_VAR

            value := _value.%B0;
        END_METHOD

        METHOD PUBLIC SetValue
            VAR_INPUT
                value: WORD;
            END_VAR

            _value := value;
        END_METHOD

        METHOD PUBLIC SetValue
            VAR_INPUT
                value: BYTE;
            END_VAR

            _value := WORD#0;
            _value.%B0 := value;
        END_METHOD
    END_CLASS

END_NAMESPACE
